(* IEC 61131-3 sources: JaccoSigma/tempclass/Class/_SCP011_111_Switch, 1 file *)

(* ---- _SCP011_111_Switch.st ---- *)
(*!
<Class
	Name               = "_SCP011_111_Switch"
	Revision           = "1.0"
	RealtimeTask       = "false"
	CyclicTask         = "false"
	BackgroundTask     = "false"
	Sigmatek           = "true"
	OSInterface        = "false"
	HighPriority       = "false"
	Automatic          = "false"
	UpdateMode         = "Prescan"
	IconPath           = ".\Class\Tool.ico"
	SharedCommandTable = "true"
	Objectsize         = "(474,120)">
	<Channels>
		<Server Name="ClassSvr" Visualized="false" Initialize="false" WriteProtected="true" Retentive="false"/>
		<Server Name="SCP011_Place" Visualized="false" Initialize="false" WriteProtected="true" Retentive="false"/>
		<Server Name="SCP111_Place" Visualized="false" Initialize="false" WriteProtected="true" Retentive="false"/>
		<Client Name="ModuleSelect" Required="true" Internal="false" Comment="Select the module used at this place&#13;&#10;0 = SCP011&#13;&#10;1 = SCP111"/>
		<Client Name="Place" Required="true" Internal="false" Comment="Place of SDIAS Modul [0..63]."/>
	</Channels>
	<RevDoku>
		<Owner Company="Sigmatek" Author="RamAnd"/>
		<Dokumentation Revision="1.0" Date="06.07.2021" Author="RamAnd" Company="Sigmatek" Description="First library version"/>
	</RevDoku>
</Class>
*)
_SCP011_111_Switch : CLASS
  //Servers:
	ClassSvr 	: SvrChCmd_DINT;
	SCP011_Place 	: SvrCh_UDINT;
	SCP111_Place 	: SvrCh_UDINT;
  //Clients:
	Place 	: CltCh_UDINT;
	ModuleSelect 	: CltCh_DINT;
  //Variables:
		bGotSelection 	: BOOL;
  //Functions:

	FUNCTION InitializePlaces;

	FUNCTION VIRTUAL GLOBAL SCP011_Place::Read
		VAR_OUTPUT
			output (EAX) 	: UDINT;
		END_VAR;

	FUNCTION VIRTUAL GLOBAL SCP111_Place::Read
		VAR_OUTPUT
			output (EAX) 	: UDINT;
		END_VAR;
  //Tables:
	FUNCTION @STD
		VAR_OUTPUT
			ret_code	: CONFSTATES;
		END_VAR;
	FUNCTION GLOBAL TAB @CT_;
END_CLASS;

FUNCTION VIRTUAL GLOBAL _SCP011_111_Switch::SCP011_Place::Read
	VAR_OUTPUT
		output (EAX) 	: UDINT;
	END_VAR

  if bGotSelection = FALSE then
    InitializePlaces();
  end_if;

	output := SCP011_Place;

END_FUNCTION

FUNCTION VIRTUAL GLOBAL _SCP011_111_Switch::SCP111_Place::Read
	VAR_OUTPUT
		output (EAX) 	: UDINT;
	END_VAR

  if bGotSelection = FALSE then
    InitializePlaces();
  end_if;

	output := SCP111_Place;

END_FUNCTION

FUNCTION _SCP011_111_Switch::InitializePlaces

  ModuleSelect := ModuleSelect.Read();
  Place          := Place.Read();

  if ModuleSelect = 0 then
    // SCP011 selected
    SCP011_Place := Place;
    SCP111_Place := DEACTIVATED_LSL;
  elsif ModuleSelect = 1 then
    // SCP111 selected
    SCP011_Place := DEACTIVATED_LSL;
    SCP111_Place := Place;
  else
    // None selected
    SCP011_Place := DEACTIVATED_LSL;
    SCP111_Place := DEACTIVATED_LSL;
  end_if;

  bGotSelection := TRUE;

END_FUNCTION
